(* PLC project Sin nombre, Desconocido Sin nombre 1 *)
(* stored: creationDateTime 2025-07-13T17:08:14, modificationDateTime 2025-07-13T20:22:26 *)

PROGRAM conexiones
  VAR
    TON0 : TON;  (* Determinar la duración de la conexión Estrella *)
    TON1 : TON;  (* Determinar la duración de la conexión Delta *)
    Pardada : BOOL;  (* Entrada del usuario para detener el sistema *)
    Conmutar : BOOL;  (* Entrada del usuario para cambiar el estado del sistema (conexion) *)
    Cambiar : BOOL;  (* Variable local para forzar el cambio de estado *)
    Detener : BOOL;  (* Variable local para interrumpir todos los procesos *)
    Delta : BOOL;  (* Determina salida para la conexion Delta *)
    Estrella : BOOL;  (* Determina salida para la conexion Estrella *)
    YOn : BOOL;  (* Encender la conexion Estrella y TON0 *)
    YOnAux : BOOL;  (* Encender la conexion Estrella y TON0 / Cuando alla cambio de estado *)
    DosOff : BOOL;  (* Apagar conexion Estrella, reiniciar TON1 y apagar TON0 *)
    DosOffAux : BOOL;  (* Apagar conexion Estrella, reiniciar TON1 y apagar TON0 /Cuando alla cambio de estado *)
    TON2 : TON;  (* Temporizador Auxiliar para remplazar TON1 *)
    TON3 : TON;  (* Temporizador Auxiliar para remplazar TON0 *)
  END_VAR

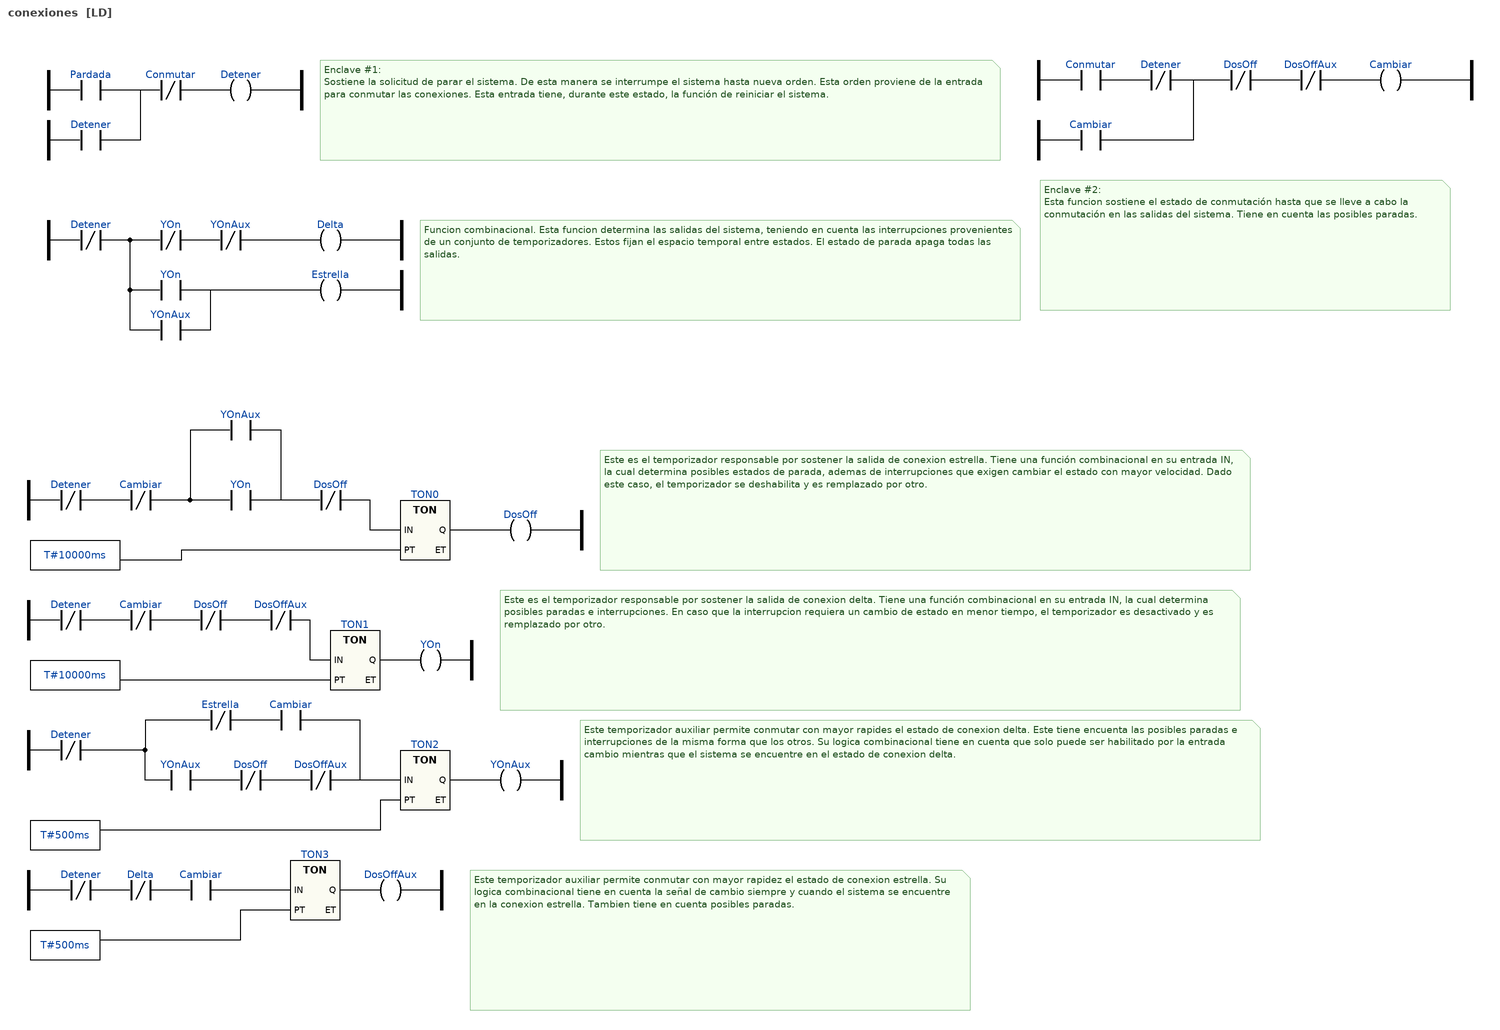
(* LD diagram, written out as Structured Text *)
(* Enclave #1:
Sostiene la solicitud de parar el sistema. De esta manera se interrumpe el sistema hasta nueva orden. Esta orden proviene de la entrada para conmutar las conexiones. Esta entrada tiene, durante este estado, la función de reiniciar el sistema. *)
Detener := (Pardada OR Detener) AND NOT Conmutar;
(* Enclave #2:
Esta funcion sostiene el estado de conmutación hasta que se lleve a cabo la conmutación en las salidas del sistema. Tiene en cuenta las posibles paradas. *)
(* Funcion combinacional. Esta funcion determina las salidas del sistema, teniendo en cuenta las interrupciones provenientes de un conjunto de temporizadores. Estos fijan el espacio temporal entre estados. El estado de parada apaga todas las salidas. *)
(* Este es el temporizador responsable por sostener la salida de conexion estrella. Tiene una función combinacional en su entrada IN, la cual determina posibles estados de parada, ademas de interrupciones que exigen cambiar el estado con mayor velocidad. Dado este caso, el temporizador se deshabilita y es remplazado por otro. *)
(* Este es el temporizador responsable por sostener la salida de conexion delta. Tiene una función combinacional en su entrada IN, la cual determina posibles paradas e interrupciones. En caso que la interrupcion requiera un cambio de estado en menor tiempo, el temporizador es desactivado y es remplazado por otro. *)
TON1(IN := NOT Detener AND NOT Cambiar AND NOT DosOff AND NOT DosOffAux, PT := T#10000ms);
YOn := TON1.Q;
TON0(IN := NOT Detener AND NOT Cambiar AND (YOn OR YOnAux) AND NOT DosOff, PT := T#10000ms);
DosOff := TON0.Q;
Delta := NOT Detener AND NOT YOn AND NOT YOnAux;
Estrella := NOT Detener AND (YOnAux OR YOn);
(* Este temporizador auxiliar permite conmutar con mayor rapides el estado de conexion delta. Este tiene encuenta las posibles paradas e interrupciones de la misma forma que los otros. Su logica combinacional tiene en cuenta que solo puede ser habilitado por la entrada cambio mientras que el sistema se encuentre en el estado de conexion delta. *)
TON2(IN := NOT Detener AND (NOT Estrella AND Cambiar OR YOnAux AND NOT DosOff AND NOT DosOffAux), PT := T#500ms);
YOnAux := TON2.Q;
(* Este temporizador auxiliar permite conmutar con mayor rapidez el estado de conexion estrella. Su logica combinacional tiene en cuenta la señal de cambio siempre y cuando el sistema se encuentre en la conexion estrella. Tambien tiene en cuenta posibles paradas. *)
TON3(IN := NOT Detener AND NOT Delta AND Cambiar, PT := T#500ms);
DosOffAux := TON3.Q;
Cambiar := (Conmutar AND NOT Detener OR Cambiar) AND NOT DosOff AND NOT DosOffAux;
END_PROGRAM

CONFIGURATION Config0
  RESOURCE Res0 ON PLC
    TASK task0(INTERVAL := T#20ms, PRIORITY := 0);
    PROGRAM instance0 WITH task0 : conexiones;
  END_RESOURCE
END_CONFIGURATION
